// TIA Portal V15.1 export
// export: Created 2024-06-21T08:41:25.6340296Z, ExportSetting WithDefaults, DisplayName Totally Integrated Automation Portal, DisplayVersion V15.1 Update 5, DisplayName TIA Portal Openness, DisplayVersion V15.1 Update 5, DisplayName SINAMICS Startdrive Advanced, DisplayVersion V15.1, DisplayName G130, G150, S120, S150, SINAMICS MV, S210, DisplayVersion V15.1, DisplayName G110M, G120, G120C, G120D, G120P, DisplayVersion V15.1, DisplayName STEP 7 Professional, DisplayVersion V15.1 Update 5, DisplayName STEP 7 Safety, DisplayVersion V15.1, DisplayName WinCC Professional, DisplayVersion V15.1 Update 5, DisplayName SIMATIC Visualization Architect, DisplayVersion V15.1
FUNCTION "209000NCP01AS" : Void   // FC294, FBD
TITLE = 209000NCP01AS Panels
{ S7_Optimized_Access := 'TRUE' }
AUTHOR : VCC
VERSION : 0.1
// stored: AutoNumber false, IsIECCheckEnabled false, SetENOAutomatically False, UDAEnableTagReadback false
   VAR_OUTPUT
      O_AlarmA : Bool;   // Alarm A
      O_AlarmB : Bool;   // Alarm B
      O_AlarmC : Bool;   // Alarm C
      O_AlarmD : Bool;   // Alarm D
      O_AlarmABCondition : Bool;   // Alarm AB condition
      H_IAnim : Word;   // For animation of icon
   END_VAR
BEGIN

REGION Network 1: **** 2.2 Alarms - Alarm generation **** 209000AS01ST1 Temperature to High
   // Temperature to High
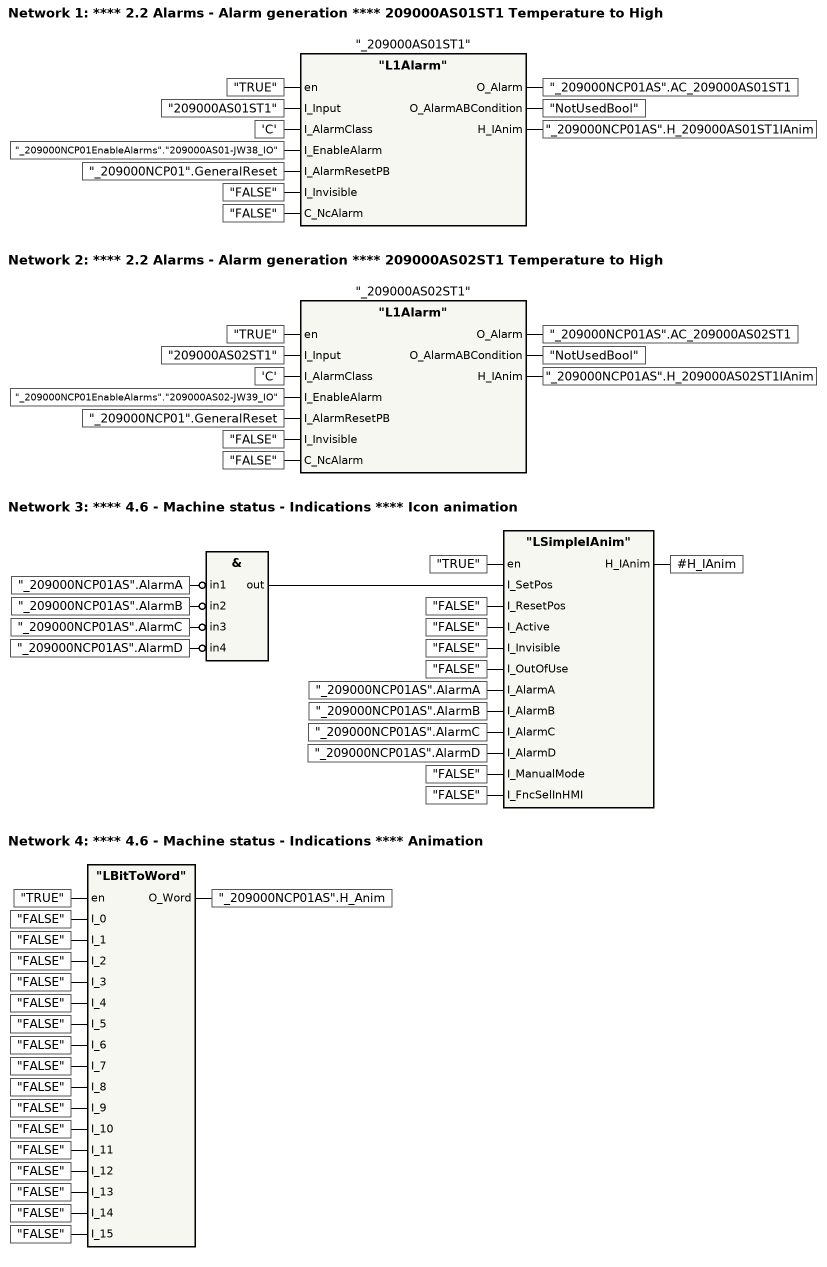
   IF "TRUE" THEN
       "_209000AS01ST1"(I_Input := "209000AS01ST1",   // "L1Alarm"
                        I_AlarmClass := 'C',
                        I_EnableAlarm := "_209000NCP01EnableAlarms"."209000AS01-JW38_IO",
                        I_AlarmResetPB := "_209000NCP01".GeneralReset,
                        I_Invisible := "FALSE",
                        C_NcAlarm := "FALSE",
                        O_Alarm => "_209000NCP01AS".AC_209000AS01ST1,
                        O_AlarmABCondition => "NotUsedBool",
                        H_IAnim => "_209000NCP01AS".H_209000AS01ST1IAnim);
   END_IF;
END_REGION

REGION Network 2: **** 2.2 Alarms - Alarm generation **** 209000AS02ST1 Temperature to High
   // Temperature to High
   IF "TRUE" THEN
       "_209000AS02ST1"(I_Input := "209000AS02ST1",   // "L1Alarm"
                        I_AlarmClass := 'C',
                        I_EnableAlarm := "_209000NCP01EnableAlarms"."209000AS02-JW39_IO",
                        I_AlarmResetPB := "_209000NCP01".GeneralReset,
                        I_Invisible := "FALSE",
                        C_NcAlarm := "FALSE",
                        O_Alarm => "_209000NCP01AS".AC_209000AS02ST1,
                        O_AlarmABCondition => "NotUsedBool",
                        H_IAnim => "_209000NCP01AS".H_209000AS02ST1IAnim);
   END_IF;
END_REGION

REGION Network 3: **** 4.6 - Machine status - Indications **** Icon animation
   // Icon animation
   IF "TRUE" THEN
       "LSimpleIAnim"(I_SetPos := NOT "_209000NCP01AS".AlarmA AND NOT "_209000NCP01AS".AlarmB AND NOT "_209000NCP01AS".AlarmC AND NOT "_209000NCP01AS".AlarmD,
                      I_ResetPos := "FALSE",
                      I_Active := "FALSE",
                      I_Invisible := "FALSE",
                      I_OutOfUse := "FALSE",
                      I_AlarmA := "_209000NCP01AS".AlarmA,
                      I_AlarmB := "_209000NCP01AS".AlarmB,
                      I_AlarmC := "_209000NCP01AS".AlarmC,
                      I_AlarmD := "_209000NCP01AS".AlarmD,
                      I_ManualMode := "FALSE",
                      I_FncSelInHMI := "FALSE",
                      H_IAnim => #H_IAnim);
   END_IF;
END_REGION

REGION Network 4: **** 4.6 - Machine status - Indications **** Animation
   // Animation
   IF "TRUE" THEN
       "LBitToWord"(I_0 := "FALSE",
                    I_1 := "FALSE",
                    I_2 := "FALSE",
                    I_3 := "FALSE",
                    I_4 := "FALSE",
                    I_5 := "FALSE",
                    I_6 := "FALSE",
                    I_7 := "FALSE",
                    I_8 := "FALSE",
                    I_9 := "FALSE",
                    I_10 := "FALSE",
                    I_11 := "FALSE",
                    I_12 := "FALSE",
                    I_13 := "FALSE",
                    I_14 := "FALSE",
                    I_15 := "FALSE",
                    O_Word => "_209000NCP01AS".H_Anim);
   END_IF;
END_REGION

NETWORK
TITLE = **** 4.6 - Machine Status - Indications **** Animation DB number
// DB number
      OPN   "_209000NCP01AS";
      L     DBNO;
      T     "_209000NCP01AS".H_DBnr;

REGION Network 6: **** 4.6 - Machine Status - Indication **** LED Indication 209000AS01 - Start/Reset
   // The Module handles indications for Start and Reset buttons
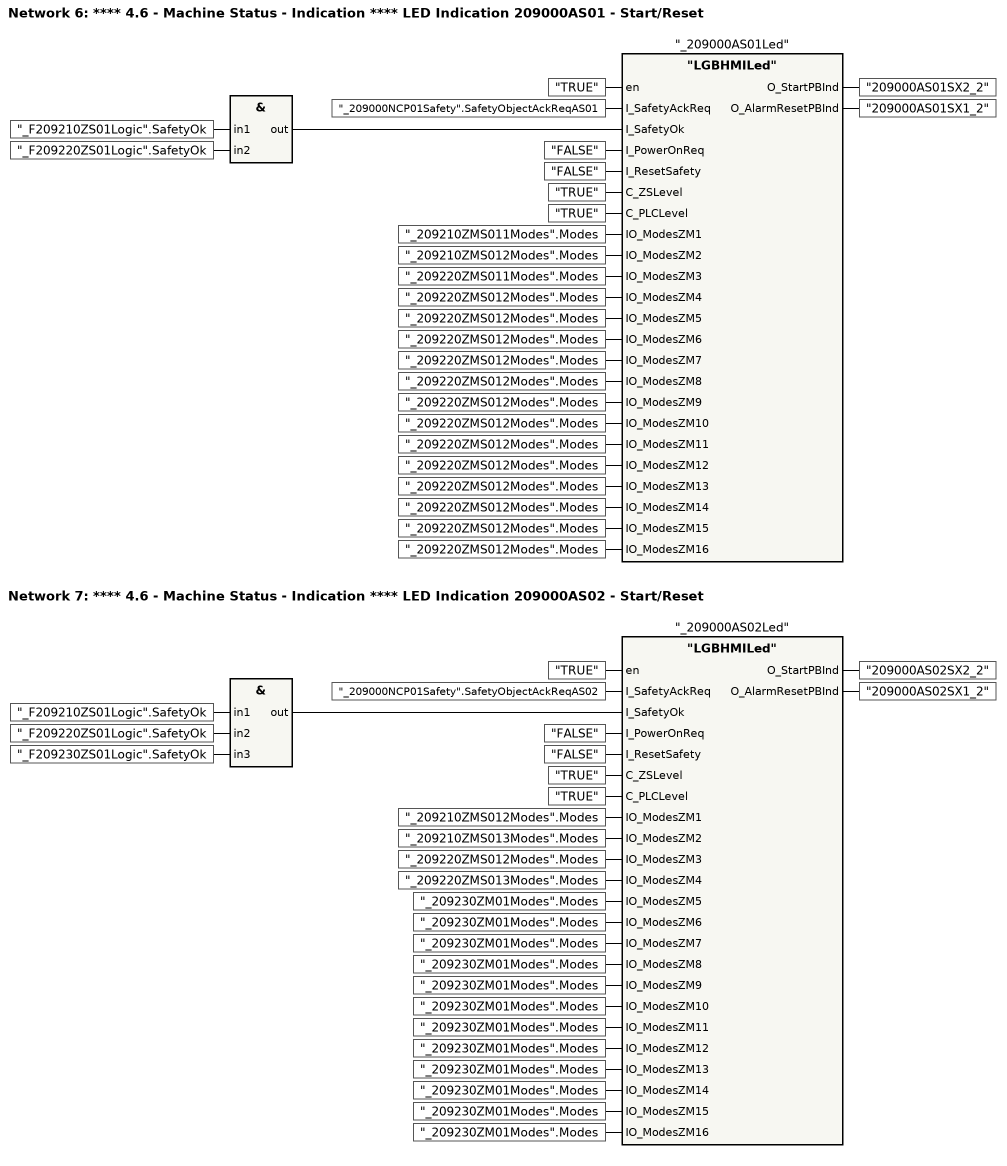
   IF "TRUE" THEN
       "_209000AS01Led"(I_SafetyAckReq := "_209000NCP01Safety".SafetyObjectAckReqAS01,   // "LGBHMILed"
                        I_SafetyOk := "_F209210ZS01Logic".SafetyOk AND "_F209220ZS01Logic".SafetyOk,
                        I_PowerOnReq := "FALSE",
                        I_ResetSafety := "FALSE",
                        C_ZSLevel := "TRUE",
                        C_PLCLevel := "TRUE",
                        IO_ModesZM1 := "_209210ZMS011Modes".Modes,
                        IO_ModesZM2 := "_209210ZMS012Modes".Modes,
                        IO_ModesZM3 := "_209220ZMS011Modes".Modes,
                        IO_ModesZM4 := "_209220ZMS012Modes".Modes,
                        IO_ModesZM5 := "_209220ZMS012Modes".Modes,
                        IO_ModesZM6 := "_209220ZMS012Modes".Modes,
                        IO_ModesZM7 := "_209220ZMS012Modes".Modes,
                        IO_ModesZM8 := "_209220ZMS012Modes".Modes,
                        IO_ModesZM9 := "_209220ZMS012Modes".Modes,
                        IO_ModesZM10 := "_209220ZMS012Modes".Modes,
                        IO_ModesZM11 := "_209220ZMS012Modes".Modes,
                        IO_ModesZM12 := "_209220ZMS012Modes".Modes,
                        IO_ModesZM13 := "_209220ZMS012Modes".Modes,
                        IO_ModesZM14 := "_209220ZMS012Modes".Modes,
                        IO_ModesZM15 := "_209220ZMS012Modes".Modes,
                        IO_ModesZM16 := "_209220ZMS012Modes".Modes,
                        O_StartPBInd => "209000AS01SX2_2",
                        O_AlarmResetPBInd => "209000AS01SX1_2");
   END_IF;
END_REGION

REGION Network 7: **** 4.6 - Machine Status - Indication **** LED Indication 209000AS02 - Start/Reset
   // The Module handles indications for Start and Reset buttons
   IF "TRUE" THEN
       "_209000AS02Led"(I_SafetyAckReq := "_209000NCP01Safety".SafetyObjectAckReqAS02,   // "LGBHMILed"
                        I_SafetyOk := "_F209210ZS01Logic".SafetyOk AND "_F209220ZS01Logic".SafetyOk AND "_F209230ZS01Logic".SafetyOk,
                        I_PowerOnReq := "FALSE",
                        I_ResetSafety := "FALSE",
                        C_ZSLevel := "TRUE",
                        C_PLCLevel := "TRUE",
                        IO_ModesZM1 := "_209210ZMS012Modes".Modes,
                        IO_ModesZM2 := "_209210ZMS013Modes".Modes,
                        IO_ModesZM3 := "_209220ZMS012Modes".Modes,
                        IO_ModesZM4 := "_209220ZMS013Modes".Modes,
                        IO_ModesZM5 := "_209230ZM01Modes".Modes,
                        IO_ModesZM6 := "_209230ZM01Modes".Modes,
                        IO_ModesZM7 := "_209230ZM01Modes".Modes,
                        IO_ModesZM8 := "_209230ZM01Modes".Modes,
                        IO_ModesZM9 := "_209230ZM01Modes".Modes,
                        IO_ModesZM10 := "_209230ZM01Modes".Modes,
                        IO_ModesZM11 := "_209230ZM01Modes".Modes,
                        IO_ModesZM12 := "_209230ZM01Modes".Modes,
                        IO_ModesZM13 := "_209230ZM01Modes".Modes,
                        IO_ModesZM14 := "_209230ZM01Modes".Modes,
                        IO_ModesZM15 := "_209230ZM01Modes".Modes,
                        IO_ModesZM16 := "_209230ZM01Modes".Modes,
                        O_StartPBInd => "209000AS02SX2_2",
                        O_AlarmResetPBInd => "209000AS02SX1_2");
   END_IF;
END_REGION

REGION Network 8: **** 4.6 - Machine Status - Indication **** Stack Light 209000AS01
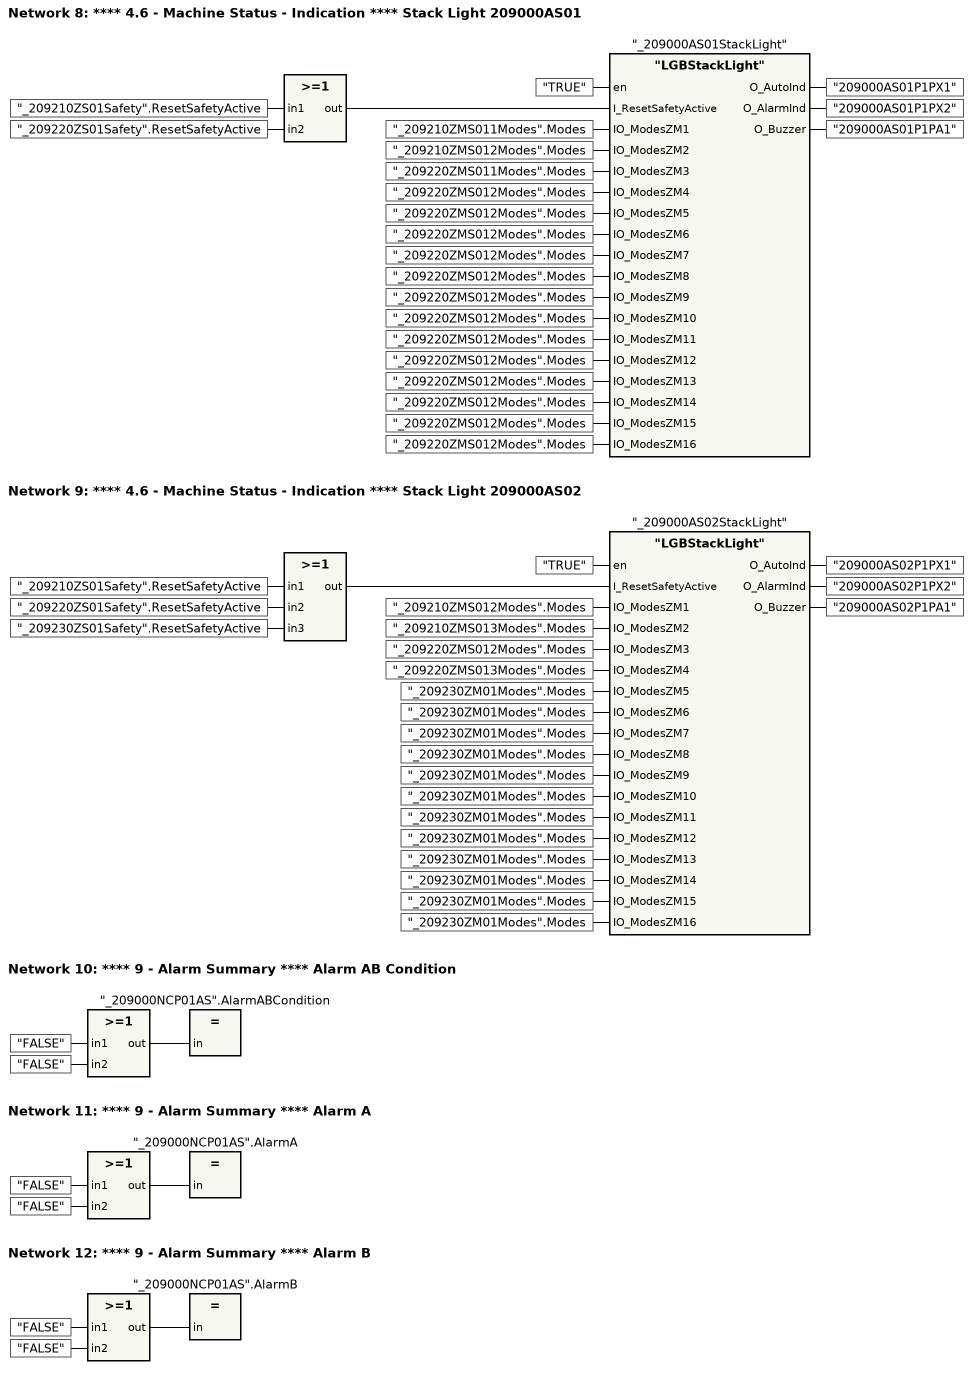
   IF "TRUE" THEN
       "_209000AS01StackLight"(I_ResetSafetyActive := "_209210ZS01Safety".ResetSafetyActive OR "_209220ZS01Safety".ResetSafetyActive,   // "LGBStackLight"
                               IO_ModesZM1 := "_209210ZMS011Modes".Modes,
                               IO_ModesZM2 := "_209210ZMS012Modes".Modes,
                               IO_ModesZM3 := "_209220ZMS011Modes".Modes,
                               IO_ModesZM4 := "_209220ZMS012Modes".Modes,
                               IO_ModesZM5 := "_209220ZMS012Modes".Modes,
                               IO_ModesZM6 := "_209220ZMS012Modes".Modes,
                               IO_ModesZM7 := "_209220ZMS012Modes".Modes,
                               IO_ModesZM8 := "_209220ZMS012Modes".Modes,
                               IO_ModesZM9 := "_209220ZMS012Modes".Modes,
                               IO_ModesZM10 := "_209220ZMS012Modes".Modes,
                               IO_ModesZM11 := "_209220ZMS012Modes".Modes,
                               IO_ModesZM12 := "_209220ZMS012Modes".Modes,
                               IO_ModesZM13 := "_209220ZMS012Modes".Modes,
                               IO_ModesZM14 := "_209220ZMS012Modes".Modes,
                               IO_ModesZM15 := "_209220ZMS012Modes".Modes,
                               IO_ModesZM16 := "_209220ZMS012Modes".Modes,
                               O_AutoInd => "209000AS01P1PX1",
                               O_AlarmInd => "209000AS01P1PX2",
                               O_Buzzer => "209000AS01P1PA1");
   END_IF;
END_REGION

REGION Network 9: **** 4.6 - Machine Status - Indication **** Stack Light 209000AS02
   IF "TRUE" THEN
       "_209000AS02StackLight"(I_ResetSafetyActive := "_209210ZS01Safety".ResetSafetyActive OR "_209220ZS01Safety".ResetSafetyActive OR "_209230ZS01Safety".ResetSafetyActive,   // "LGBStackLight"
                               IO_ModesZM1 := "_209210ZMS012Modes".Modes,
                               IO_ModesZM2 := "_209210ZMS013Modes".Modes,
                               IO_ModesZM3 := "_209220ZMS012Modes".Modes,
                               IO_ModesZM4 := "_209220ZMS013Modes".Modes,
                               IO_ModesZM5 := "_209230ZM01Modes".Modes,
                               IO_ModesZM6 := "_209230ZM01Modes".Modes,
                               IO_ModesZM7 := "_209230ZM01Modes".Modes,
                               IO_ModesZM8 := "_209230ZM01Modes".Modes,
                               IO_ModesZM9 := "_209230ZM01Modes".Modes,
                               IO_ModesZM10 := "_209230ZM01Modes".Modes,
                               IO_ModesZM11 := "_209230ZM01Modes".Modes,
                               IO_ModesZM12 := "_209230ZM01Modes".Modes,
                               IO_ModesZM13 := "_209230ZM01Modes".Modes,
                               IO_ModesZM14 := "_209230ZM01Modes".Modes,
                               IO_ModesZM15 := "_209230ZM01Modes".Modes,
                               IO_ModesZM16 := "_209230ZM01Modes".Modes,
                               O_AutoInd => "209000AS02P1PX1",
                               O_AlarmInd => "209000AS02P1PX2",
                               O_Buzzer => "209000AS02P1PA1");
   END_IF;
END_REGION

REGION Network 10: **** 9 - Alarm Summary **** Alarm AB Condition
   // Alarm AB condition
   "_209000NCP01AS".AlarmABCondition := "FALSE" OR "FALSE";
END_REGION

REGION Network 11: **** 9 - Alarm Summary **** Alarm A
   // Summary of alarms A
   "_209000NCP01AS".AlarmA := "FALSE" OR "FALSE";
END_REGION

REGION Network 12: **** 9 - Alarm Summary **** Alarm B
   // Summary of alarms B
   "_209000NCP01AS".AlarmB := "FALSE" OR "FALSE";
END_REGION

REGION Network 13: **** 9 - Alarm Summary **** Alarm C
   // Summary of alarms C
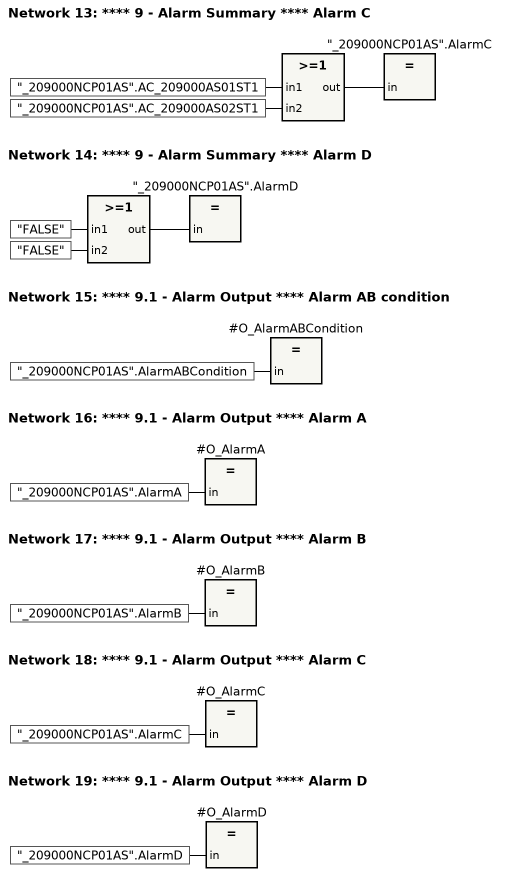
   "_209000NCP01AS".AlarmC := "_209000NCP01AS".AC_209000AS01ST1 OR "_209000NCP01AS".AC_209000AS02ST1;
END_REGION

REGION Network 14: **** 9 - Alarm Summary **** Alarm D
   // Summary of alarms D
   "_209000NCP01AS".AlarmD := "FALSE" OR "FALSE";
END_REGION

REGION Network 15: **** 9.1 - Alarm Output **** Alarm AB condition
   // Alarm AB condition
   #O_AlarmABCondition := "_209000NCP01AS".AlarmABCondition;
END_REGION

REGION Network 16: **** 9.1 - Alarm Output **** Alarm A
   // Output Alarm A
   #O_AlarmA := "_209000NCP01AS".AlarmA;
END_REGION

REGION Network 17: **** 9.1 - Alarm Output **** Alarm B
   // Output Alarm B
   #O_AlarmB := "_209000NCP01AS".AlarmB;
END_REGION

REGION Network 18: **** 9.1 - Alarm Output **** Alarm C
   // Output Alarm A
   #O_AlarmC := "_209000NCP01AS".AlarmC;
END_REGION

REGION Network 19: **** 9.1 - Alarm Output **** Alarm D
   // Output Alarm D
   #O_AlarmD := "_209000NCP01AS".AlarmD;
END_REGION

REGION Network 20: **** 9.2 - Alarm DWord**** Alarm To DWord
   // Alarm Word
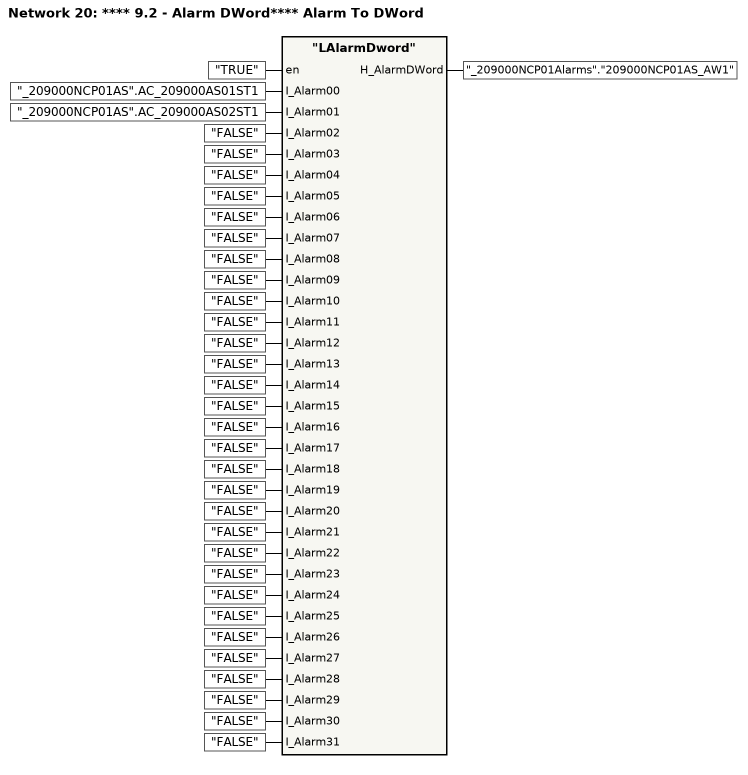
   IF "TRUE" THEN
       "LAlarmDword"(I_Alarm00 := "_209000NCP01AS".AC_209000AS01ST1,
                     I_Alarm01 := "_209000NCP01AS".AC_209000AS02ST1,
                     I_Alarm02 := "FALSE",
                     I_Alarm03 := "FALSE",
                     I_Alarm04 := "FALSE",
                     I_Alarm05 := "FALSE",
                     I_Alarm06 := "FALSE",
                     I_Alarm07 := "FALSE",
                     I_Alarm08 := "FALSE",
                     I_Alarm09 := "FALSE",
                     I_Alarm10 := "FALSE",
                     I_Alarm11 := "FALSE",
                     I_Alarm12 := "FALSE",
                     I_Alarm13 := "FALSE",
                     I_Alarm14 := "FALSE",
                     I_Alarm15 := "FALSE",
                     I_Alarm16 := "FALSE",
                     I_Alarm17 := "FALSE",
                     I_Alarm18 := "FALSE",
                     I_Alarm19 := "FALSE",
                     I_Alarm20 := "FALSE",
                     I_Alarm21 := "FALSE",
                     I_Alarm22 := "FALSE",
                     I_Alarm23 := "FALSE",
                     I_Alarm24 := "FALSE",
                     I_Alarm25 := "FALSE",
                     I_Alarm26 := "FALSE",
                     I_Alarm27 := "FALSE",
                     I_Alarm28 := "FALSE",
                     I_Alarm29 := "FALSE",
                     I_Alarm30 := "FALSE",
                     I_Alarm31 := "FALSE",
                     H_AlarmDWord => "_209000NCP01Alarms"."209000NCP01AS_AW1");
   END_IF;
END_REGION
END_FUNCTION
